// TIA Portal V19 export
FUNCTION_BLOCK "ButtonsSafe_LB113_W"   // FB46, LAD
TITLE = LB1.2 SAFE BUTTONS (@ Straightener entry)
// stored: MemoryReserve 100, SetENOAutomatically false
   VAR_INPUT
      Reset_OthersPBs_Activation_IN : Bool := FALSE;
   END_VAR
   VAR_OUTPUT
      Reset_OthersPBs_Activation_OUT : Bool;
   END_VAR
   VAR
      i : Int;
      iOperation : Int;
      iConcurrentOperation : Int;
      SettingWriteDone : Bool;
      PbPanel : "Buttons2Hands";
      PB : Struct
         ResetAlarms : Bool;
         JBTorch_Fwd : Bool;
         JBTorch_Bwd : Bool;
         JBWeldMan : Bool;
      END_STRUCT;
   END_VAR
   VAR CONSTANT
      ITEMS : Int := 3;
      TORCH_FWD : Int := 1;
      TORCH_BWD : Int := 2;
      WELD_MAN : Int := 3;
   END_VAR
BEGIN

REGION Network 1 (SCL): Interlocks between operations selected
   IF "Area01".AreaInterface.ManOneShot THEN
       #SettingWriteDone := FALSE;
   END_IF;

   // Interblocco tra operazioni
   // 
   IF NOT #SettingWriteDone THEN
       #SettingWriteDone := TRUE;

       FOR #iOperation := 1 TO #ITEMS DO
           FOR #iConcurrentOperation := 1 TO #ITEMS DO
               #PbPanel.Enables[#iOperation, #iConcurrentOperation] := FALSE;
           END_FOR;
       END_FOR;


       #PbPanel.Enables[TORCH_FWD, WELD_MAN] := TRUE;

       #PbPanel.Enables[WELD_MAN, TORCH_FWD] := TRUE;

   END_IF;
END_REGION

REGION Network 2 (SCL): Buttons for Op selection
   #PbPanel.Buttons[TORCH_FWD] := "LB113_JB_Torch_Pb_Fwd";
   #PbPanel.Buttons[TORCH_BWD] := "LB113_JB_Torch_Pb_Bwd";
   #PbPanel.Buttons[WELD_MAN] := "LB113_JB_Weld_Pb_Man";
END_REGION

REGION Network 3 (SCL): Operation enable

   #PbPanel.OpEnabled[TORCH_FWD] := "JB".COut.Torch.PlusCheckNext;
   #PbPanel.OpEnabled[TORCH_BWD] := "JB".COut.Torch.MinusCheckNext;

   #PbPanel.OpEnabled[WELD_MAN] := "JB".COut.Weld_CheckNext;
END_REGION

REGION Network 4 (SCL): Operation running

   #PbPanel.OpRunning[TORCH_FWD] := "JB".COut.Torch.PlusRunning;
   #PbPanel.OpRunning[TORCH_BWD] := "JB".COut.Torch.MinusRunning;

   #PbPanel.OpRunning[WELD_MAN] := "JB".DataOut.WelderON;
END_REGION

REGION Network 5 (SCL): Operation done
   #PbPanel.OpDone[TORCH_FWD] := "JB".COut.Torch.PlusLimitReached;
   #PbPanel.OpDone[TORCH_BWD] := "JB".COut.Torch.MinusLimitReached;

   #PbPanel.OpDone[WELD_MAN] := FALSE;
END_REGION

REGION Network 6: Main
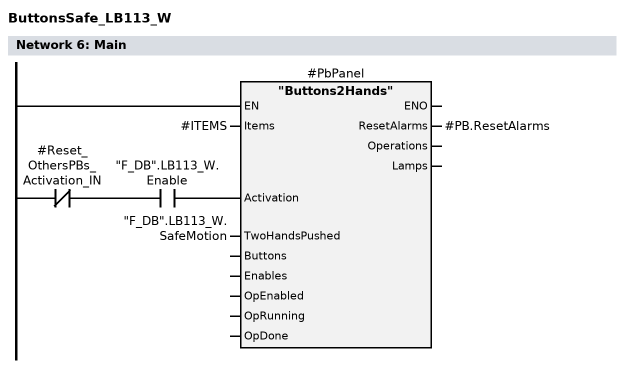
   RUNG wire#powerrail
      #PbPanel(Activation := wire#w1, Items := #ITEMS, TwoHandsPushed := "F_DB".LB113_W.SafeMotion, Buttons :=, Enables :=, OpEnabled :=, OpRunning :=, OpDone :=, ResetAlarms => #PB.ResetAlarms, Operations =>, Lamps =>)
   END_RUNG
   RUNG wire#powerrail
      I_Contact( #Reset_OthersPBs_Activation_IN )
      Contact( "F_DB".LB113_W.Enable )
   END_RUNG wire#w1
   // the same network as SCL:
   #PbPanel(Items := #ITEMS,   // "Buttons2Hands"
            Activation := NOT #Reset_OthersPBs_Activation_IN AND "F_DB".LB113_W.Enable,
            TwoHandsPushed := "F_DB".LB113_W.SafeMotion,
            ResetAlarms => #PB.ResetAlarms);
END_REGION

REGION Network 7 (SCL): Safe Buttons
   #PB.JBTorch_Fwd := #PbPanel.Operations[TORCH_FWD];
   #PB.JBTorch_Bwd := #PbPanel.Operations[TORCH_BWD];
   #PB.JBWeldMan := #PbPanel.Operations[WELD_MAN];
END_REGION

REGION Network 8 (SCL): Lamp selection

   "LB113_JB_Torch_Lp_Fwd" := #PbPanel.Lamps[TORCH_FWD];
   "LB113_JB_Torch_Lp_Bwd" := #PbPanel.Lamps[TORCH_BWD];

   "LB113_JB_Weld_Lp_Man" := #PbPanel.Lamps[WELD_MAN];
END_REGION

REGION Network 9 (SCL): Reset others safe push buttons activation / execution
   #Reset_OthersPBs_Activation_OUT := FALSE;

   FOR #i := 1 TO #ITEMS DO

       IF #PbPanel.Buttons[#i] OR #PbPanel.Operations[#i] THEN
           #Reset_OthersPBs_Activation_OUT := TRUE;
           EXIT;
       END_IF;

   END_FOR;
END_REGION

REGION Network 10: >
END_REGION

REGION Network 11: >
END_REGION

REGION Network 12: >
END_REGION
END_FUNCTION_BLOCK
